// TIA Portal V20 export
TYPE "typeSequenceControlNode_sideTapeFixStage"
// stored: Namespace Unit1.Em4
   STRUCT
      jobs : "LAF_typeJobs";
      sequence : "LAF_typeSequence";
      selectJobStatus { S7_SetPoint := 'True'} : Array[0..10] of "LAF_typeJobStatus";
      "step" : "LER_typeStep";
      jobInterface : "Unit1.Em4.typeSequenceControlNodeJobInterface_sideTapeFixStage";
      homeCheck : "Unit1.Em4.typeSequenceControlNodeHomeCheck_sideTapeFixStage";
   END_STRUCT;
   // // "step".action1[101] : Step[101] : JOB[1] Condition
   // // "step".action1[110] : Step[110] : Side Tape Fix Stage Clamp Open
   // // "step".action1[111] : Step[111] : Side Tape Fix Stage Clamp Close
   // // "step".action1[120] : Step[120] : Side Tape Fix Stage X-Axis JR Get Pos
   // // "step".action1[130] : Step[130] : Side Tape Fix Stage C-Axis Wait Pos [Tape-1]
   // // "step".action1[131] : Step[131] : Side Tape Fix Stage C-Axis Tape-2 Pos
   // // "step".action1[132] : Step[132] : Side Tape Fix Stage C-Axis Tape-3 Pos
   // // "step".action1[133] : Step[133] : Side Tape Fix Stage C-Axis Tape-4 Pos
   // // "step".action1[140] : Step[140] : Side Tape Fix Stage X-Axis Wait Pos
   // // "step".action1[190] : Step[190] : JOB[1] Step End
   // // "step".action1[201] : Step[201] : JOB[2] Condition
   // // "step".action1[210] : Step[210] : Side Tape Fix Stage [Loading Request] => JR PP Right
   // // "step".action1[220] : Step[220] : Side Tape Fix Stage X-Axis JR Get Pos
   // // "step".action1[230] : Step[230] : Side Tape Fix Stage Clamp Close
   // // "step".action1[231] : Step[231] : Data Transfer
   // // "step".action1[232] : Step[232] : Side Tape Fix Stage [Unclamp Request] => JR PP Right
   // // "step".action1[280] : Step[280] : Side Tape Fix Stage X-Axis Wait Pos
   // // "step".action1[290] : Step[290] : JOB[2] Step End
   // // "step".action1[301] : Step[301] : JOB[4] Condition
   // // "step".action1[310] : Step[310] : Spare
   // // "step".action1[320] : Step[320] : Side Tape Fix Stage => Call Attachment Tape-1
   // // "step".action1[390] : Step[390] : JOB[3] Step End
   // // "step".action1[401] : Step[401] : JOB[4] Condition
   // // "step".action1[410] : Step[410] : Side Tape Fix Stage X-Axis Wait Pos
   // // "step".action1[411] : Step[411] : Side Tape Fix Stage C-Axis Taping-2 Pos
   // // "step".action1[412] : Step[412] : Side Tape Fix Stage X-Axis Wait Pos
   // // "step".action1[420] : Step[420] : Side Tape Fix Stage => Call Attachment Tape-2
   // // "step".action1[490] : Step[490] : JOB[4] Step End
   // // "step".action1[501] : Step[501] : JOB[5] Condition
   // // "step".action1[510] : Step[510] : Side Tape Fix Stage X-Axis Wait Pos
   // // "step".action1[511] : Step[511] : Side Tape Fix Stage C-Axis Taping-3 Pos
   // // "step".action1[512] : Step[512] : Side Tape Fix Stage X-Axis Wait Pos
   // // "step".action1[520] : Step[520] : Side Tape Fix Stage => Call Attachment Tape-3
   // // "step".action1[590] : Step[590] : JOB[5] Step End
   // // "step".action1[601] : Step[601] : JOB[6] Condition
   // // "step".action1[610] : Step[610] : Side Tape Fix Stage X-Axis Wait Pos
   // // "step".action1[611] : Step[611] : Side Tape Fix Stage C-Axis Taping-4 Pos
   // // "step".action1[612] : Step[612] : Side Tape Fix Stage X-Axis Wait Pos
   // // "step".action1[620] : Step[620] : Side Tape Fix Stage => Call Attachment Tape-4
   // // "step".action1[690] : Step[690] : JOB[6] Step End
   // // "step".action1[701] : Step[701] : JOB[7] Condition
   // // "step".action1[710] : Step[710] : Side Tape Fix Stage X-Axis Put Pos
   // // "step".action1[720] : Step[720] : Side Tape Fix Stage [Unloading Request] => Transfer PP Left
   // // "step".action1[721] : Step[721] : Side Tape Fix Stage [Clamp Request] => Transfer PP Left
   // // "step".action1[722] : Step[722] : Side Tape Fix Stage Clamp Open
   // // "step".action1[723] : Step[723] : Side Tape Fix Stage [Backward Request] => Transfer PP Left
   // // "step".action1[780] : Step[780] : Side Tape Fix Stage X-Axis Wait Pos
   // // "step".action1[781] : Step[781] : Side Tape Fix Stage C-Axis Wait Pos
   // // "step".action1[782] : Step[782] : Side Tape Fix Stage X-Axis Wait Pos
   // // "step".action1[790] : Step[790] : JOB[7] Step End
   // // "step".transition1[101] : Step[101] : JOB[1] Condition
   // // "step".transition1[110] : Step[110] : Side Tape Fix Stage Clamp Open
   // // "step".transition1[111] : Step[111] : Side Tape Fix Stage Clamp Close
   // // "step".transition1[120] : Step[120] : Side Tape Fix Stage X-Axis JR Get Pos
   // // "step".transition1[130] : Step[130] : Side Tape Fix Stage C-Axis Wait Pos [Tape-1]
   // // "step".transition1[131] : Step[131] : Side Tape Fix Stage C-Axis Tape-2 Pos
   // // "step".transition1[132] : Step[132] : Side Tape Fix Stage C-Axis Tape-3 Pos
   // // "step".transition1[133] : Step[133] : Side Tape Fix Stage C-Axis Tape-4 Pos
   // // "step".transition1[140] : Step[140] : Side Tape Fix Stage X-Axis Wait Pos
   // // "step".transition1[190] : Step[190] : JOB[1] Step End
   // // "step".transition1[201] : Step[201] : JOB[2] Condition
   // // "step".transition1[210] : Step[210] : Side Tape Fix Stage [Loading Request] => JR PP Right
   // // "step".transition1[220] : Step[220] : Side Tape Fix Stage X-Axis JR Get Pos
   // // "step".transition1[230] : Step[230] : Side Tape Fix Stage Clamp Close
   // // "step".transition1[231] : Step[231] : Data Transfer
   // // "step".transition1[232] : Step[232] : Side Tape Fix Stage [Unclamp Request] => JR PP Right
   // // "step".transition1[280] : Step[280] : Side Tape Fix Stage X-Axis Wait Pos
   // // "step".transition1[290] : Step[290] : JOB[2] Step End
   // // "step".transition1[301] : Step[301] : JOB[4] Condition
   // // "step".transition1[310] : Step[310] : Spare
   // // "step".transition1[320] : Step[320] : Side Tape Fix Stage => Call Attachment Tape-1
   // // "step".transition1[390] : Step[390] : JOB[3] Step End
   // // "step".transition1[401] : Step[401] : JOB[4] Condition
   // // "step".transition1[410] : Step[410] : Side Tape Fix Stage X-Axis Wait Pos
   // // "step".transition1[411] : Step[411] : Side Tape Fix Stage C-Axis Taping-2 Pos
   // // "step".transition1[412] : Step[412] : Side Tape Fix Stage X-Axis Wait Pos
   // // "step".transition1[420] : Step[420] : Side Tape Fix Stage => Call Attachment Tape-2
   // // "step".transition1[490] : Step[490] : JOB[4] Step End
   // // "step".transition1[501] : Step[501] : JOB[5] Condition
   // // "step".transition1[510] : Step[510] : Side Tape Fix Stage X-Axis Wait Pos
   // // "step".transition1[511] : Step[511] : Side Tape Fix Stage C-Axis Taping-3 Pos
   // // "step".transition1[512] : Step[512] : Side Tape Fix Stage X-Axis Wait Pos
   // // "step".transition1[520] : Step[520] : Side Tape Fix Stage => Call Attachment Tape-3
   // // "step".transition1[590] : Step[590] : JOB[5] Step End
   // // "step".transition1[601] : Step[601] : JOB[6] Condition
   // // "step".transition1[610] : Step[610] : Side Tape Fix Stage X-Axis Wait Pos
   // // "step".transition1[611] : Step[611] : Side Tape Fix Stage C-Axis Taping-4 Pos
   // // "step".transition1[612] : Step[612] : Side Tape Fix Stage X-Axis Wait Pos
   // // "step".transition1[620] : Step[620] : Side Tape Fix Stage => Call Attachment Tape-4
   // // "step".transition1[690] : Step[690] : JOB[6] Step End
   // // "step".transition1[701] : Step[701] : JOB[7] Condition
   // // "step".transition1[710] : Step[710] : Side Tape Fix Stage X-Axis Put Pos
   // // "step".transition1[720] : Step[720] : Side Tape Fix Stage [Unloading Request] => Transfer PP Left
   // // "step".transition1[721] : Step[721] : Side Tape Fix Stage [Clamp Request] => Transfer PP Left
   // // "step".transition1[722] : Step[722] : Side Tape Fix Stage Clamp Open
   // // "step".transition1[723] : Step[723] : Side Tape Fix Stage [Backward Request] => Transfer PP Left
   // // "step".transition1[780] : Step[780] : Side Tape Fix Stage X-Axis Wait Pos
   // // "step".transition1[781] : Step[781] : Side Tape Fix Stage C-Axis Wait Pos
   // // "step".transition1[782] : Step[782] : Side Tape Fix Stage X-Axis Wait Pos
   // // "step".transition1[790] : Step[790] : JOB[7] Step End
END_TYPE
